(* IEC 61131-3 sources: OpenPLC_test_bench/Arduino_UNO/OpenPLC_LD/Bench_shield_test, 2 files *)

(* ---- Spresense_Blink.st ---- *)
PROGRAM Blink
  VAR
    blink_led AT %QX0.0 : BOOL;
  END_VAR
  VAR
    TON0 : TON;
    TOF0 : TOF;
  END_VAR

  TON0(EN := TRUE, IN := NOT(blink_led), PT := T#500ms);
  TOF0(EN := TON0.ENO, IN := TON0.Q, PT := T#500ms);
  blink_led := TOF0.Q;
END_PROGRAM

CONFIGURATION Config0

  RESOURCE Res0 ON PLC
    TASK task0(INTERVAL := T#20ms,PRIORITY := 0);
    PROGRAM instance0 WITH task0 : Blink;
  END_RESOURCE
END_CONFIGURATION

(* ---- Spresense_Blink_01.st ---- *)
PROGRAM Blink
  VAR
    blink_led AT %QX0.0 : BOOL;
    blink_led0 AT %QX100.1 : BOOL;
  END_VAR
  VAR
    TON0 : TON;
    TOF0 : TOF;
  END_VAR

  TON0(EN := TRUE, IN := NOT(blink_led), PT := T#500ms);
  TOF0(EN := TON0.ENO, IN := TON0.Q, PT := T#500ms);
  blink_led := TOF0.Q;
  blink_led0 := TOF0.Q;
END_PROGRAM

CONFIGURATION Config0

  RESOURCE Res0 ON PLC
    TASK task0(INTERVAL := T#20ms,PRIORITY := 0);
    PROGRAM instance0 WITH task0 : Blink;
  END_RESOURCE
END_CONFIGURATION
